FUNCTION_BLOCK FB_TemperatureSensor EXTENDS FB_Sensor
VAR_INPUT
END_VAR
VAR_OUTPUT
	fTemperature : REAL; //measured temperature in °C
END_VAR
VAR
	//I/O-Links
	temperature_IN AT %I* : INT;
	
END_VAR

METHOD GetState_AI : BOOL
VAR_INPUT
END_VAR
fTemperature := (temperature_IN / 32767.0)*50.0;  //conversion: scaled to temperature 0-50 °C from 0 - 10 V

//sensor state
sensorState.fValue := fTemperature;
sensorState.sUnit := 'degreeC';
END_METHOD

END_FUNCTION_BLOCK

(* stored: Version 1.1.0.1, ProductVersion 3.1.4024.6
   POU FB_TemperatureSensor: Id {a8453651-dd5f-4033-8f9b-1f0387395629}, SpecialFunc None
   Method GetState_AI: Id {e2bef95d-9f4b-49d2-9a05-4a967107124d} *)
